SUBAPPLICATION Uebung_033 (* LED Strip Blinkende LED *)
  (* Standard: 61499-2 *)
  (* Version 1.0, 2023-10-23, franz *)
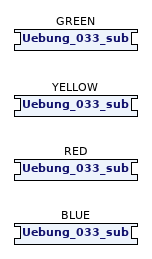
  SUBAPPS
    GREEN : Uebung_033_sub;
    YELLOW : Uebung_033_sub;
    RED : Uebung_033_sub;
    BLUE : Uebung_033_sub;
  END_SUBAPPS
END_SUBAPPLICATION
